TYPE ST_BeamParams :
STRUCT
	// Beam parameters
	// These must be filled in by the caller.
	
	//Note: fAtt is a local parameter, meaning it is distributed to the nearest
	// upstream attenuator component.
	fAtt : REAL := 100; //Requested attenuation %
	
	
	
	//Machine parameters
	nBeamClass	:	BYTE := 16#F;
	nRate	:	UDINT	:= 10; //Pulse-rate
	fPP_mJ : REAL := 20; //Per pulse max energy (mJ)
	//1.5-0keV subdivided per bit
	(*
	0.0-0.2 - 0
	0.2-0.3 - 1
	0.3-0.4 - 2
	0.4-0.5 - 3
	0.5-0.6 - 4
	0.6-0.7 - 5
	0.7-0.8 - 6
	0.8-0.9 - 7
	0.9-1.0 - 8
	1.0-1.1 - 9
	1.1-1.2 - 10
	1.2-1.3 - 11
	1.3-1.4 - 12
	1.4-1.5 - 13
	na - 14
	na - 15
	*)
	
	{attribute 'displaymode':='binary'}
	neVReqRange	:	WORD	:= 2#1111_1111_1111_1111; //Valid photon energy ranges
	
	reV	:	REAL	:=0; //Photon energy (calculated by undulator gap)

END_STRUCT
END_TYPE

(* stored: Version 1.1.0.1, ProductVersion 3.1.4022.12
   DUT ST_BeamParams: Id {1cfc4571-cdd9-4483-b0d1-cbcb7d03cd4c} *)
